// TIA Portal V19 export
FUNCTION "FC902_SafetyLogic" : Void   // FC902, F_LAD
{ S7_Optimized_Access := 'TRUE' }
// stored: AutoNumber false
BEGIN

REGION Network 1: Safety enabled to Robot Safemove
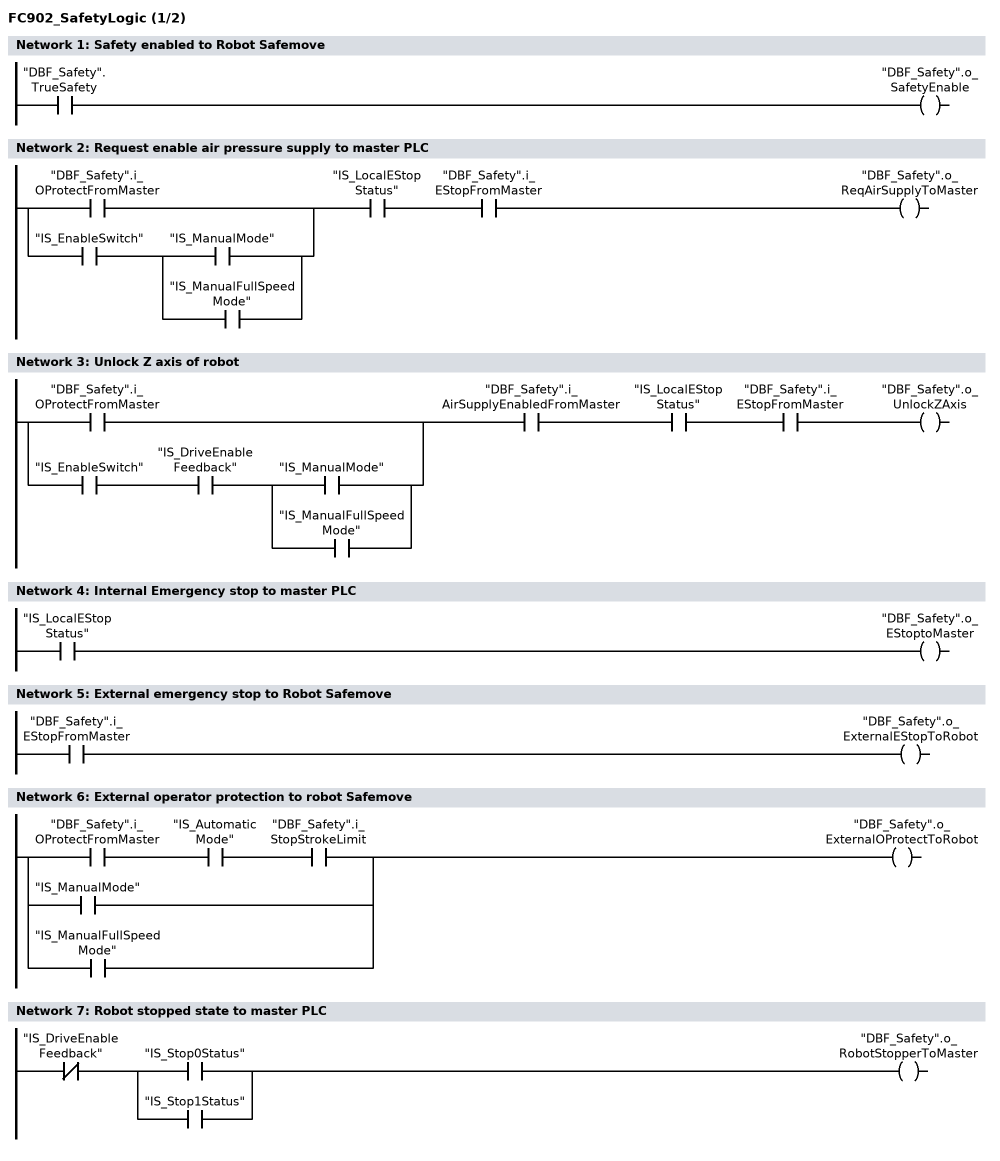
   RUNG wire#powerrail
      Contact( "DBF_Safety".TrueSafety )
      Coil( "DBF_Safety".o_SafetyEnable )
   END_RUNG
   // the same network as SCL:
   "DBF_Safety".o_SafetyEnable := "DBF_Safety".TrueSafety;
END_REGION

REGION Network 2: Request enable air pressure supply to master PLC
   RUNG wire#powerrail
      Contact( "DBF_Safety".i_OProtectFromMaster )
      wire#w1
      Contact( "IS_LocalEStopStatus" )
      Contact( "DBF_Safety".i_EStopFromMaster )
      Coil( "DBF_Safety".o_ReqAirSupplyToMaster )
   END_RUNG
   RUNG wire#powerrail
      Contact( "IS_EnableSwitch" )
      wire#w2
      Contact( "IS_ManualMode" )
   END_RUNG wire#w1
   RUNG wire#w2
      Contact( "IS_ManualFullSpeedMode" )
   END_RUNG wire#w1
   // the same network as SCL:
   "DBF_Safety".o_ReqAirSupplyToMaster := ("DBF_Safety".i_OProtectFromMaster OR ("IS_EnableSwitch" AND ("IS_ManualMode" OR "IS_ManualFullSpeedMode"))) AND "IS_LocalEStopStatus" AND "DBF_Safety".i_EStopFromMaster;
END_REGION

REGION Network 3: Unlock Z axis of robot
   RUNG wire#powerrail
      Contact( "DBF_Safety".i_OProtectFromMaster )
      wire#w1
      Contact( "DBF_Safety".i_AirSupplyEnabledFromMaster )
      Contact( "IS_LocalEStopStatus" )
      Contact( "DBF_Safety".i_EStopFromMaster )
      Coil( "DBF_Safety".o_UnlockZAxis )
   END_RUNG
   RUNG wire#powerrail
      Contact( "IS_EnableSwitch" )
      Contact( "IS_DriveEnableFeedback" )
      wire#w2
      Contact( "IS_ManualMode" )
   END_RUNG wire#w1
   RUNG wire#w2
      Contact( "IS_ManualFullSpeedMode" )
   END_RUNG wire#w1
   // the same network as SCL:
   "DBF_Safety".o_UnlockZAxis := ("DBF_Safety".i_OProtectFromMaster OR ("IS_EnableSwitch" AND "IS_DriveEnableFeedback" AND ("IS_ManualMode" OR "IS_ManualFullSpeedMode"))) AND "DBF_Safety".i_AirSupplyEnabledFromMaster AND "IS_LocalEStopStatus" AND "DBF_Safety".i_EStopFromMaster;
END_REGION

REGION Network 4: Internal Emergency stop to master PLC
   RUNG wire#powerrail
      Contact( "IS_LocalEStopStatus" )
      Coil( "DBF_Safety".o_EStoptoMaster )
   END_RUNG
   // the same network as SCL:
   "DBF_Safety".o_EStoptoMaster := "IS_LocalEStopStatus";
END_REGION

REGION Network 5: External emergency stop to Robot Safemove
   RUNG wire#powerrail
      Contact( "DBF_Safety".i_EStopFromMaster )
      Coil( "DBF_Safety".o_ExternalEStopToRobot )
   END_RUNG
   // the same network as SCL:
   "DBF_Safety".o_ExternalEStopToRobot := "DBF_Safety".i_EStopFromMaster;
END_REGION

REGION Network 6: External operator protection to robot Safemove
   RUNG wire#powerrail
      Contact( "DBF_Safety".i_OProtectFromMaster )
      Contact( "IS_AutomaticMode" )
      Contact( "DBF_Safety".i_StopStrokeLimit )
      wire#w1
      Coil( "DBF_Safety".o_ExternalOProtectToRobot )
   END_RUNG
   RUNG wire#powerrail
      Contact( "IS_ManualMode" )
   END_RUNG wire#w1
   RUNG wire#powerrail
      Contact( "IS_ManualFullSpeedMode" )
   END_RUNG wire#w1
   // the same network as SCL:
   "DBF_Safety".o_ExternalOProtectToRobot := ("DBF_Safety".i_OProtectFromMaster AND "IS_AutomaticMode" AND "DBF_Safety".i_StopStrokeLimit) OR "IS_ManualMode" OR "IS_ManualFullSpeedMode";
END_REGION

REGION Network 7: Robot stopped state to master PLC
   RUNG wire#powerrail
      I_Contact( "IS_DriveEnableFeedback" )
      wire#w1
      Contact( "IS_Stop0Status" )
      wire#w2
      Coil( "DBF_Safety".o_RobotStopperToMaster )
   END_RUNG
   RUNG wire#w1
      Contact( "IS_Stop1Status" )
   END_RUNG wire#w2
   // the same network as SCL:
   "DBF_Safety".o_RobotStopperToMaster := NOT "IS_DriveEnableFeedback" AND ("IS_Stop0Status" OR "IS_Stop1Status");
END_REGION

REGION Network 8: Power Off 24V Safety for FerRobotic
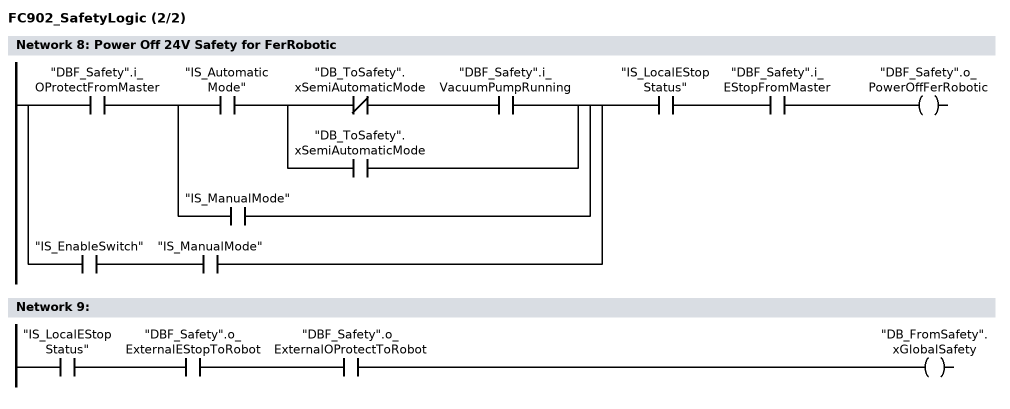
   RUNG wire#powerrail
      Contact( "DBF_Safety".i_OProtectFromMaster )
      wire#w1
      Contact( "IS_AutomaticMode" )
      wire#w2
      I_Contact( "DB_ToSafety".xSemiAutomaticMode )
      Contact( "DBF_Safety".i_VacuumPumpRunning )
      wire#w3
      Contact( "IS_LocalEStopStatus" )
      Contact( "DBF_Safety".i_EStopFromMaster )
      Coil( "DBF_Safety".o_PowerOffFerRobotic )
   END_RUNG
   RUNG wire#w2
      Contact( "DB_ToSafety".xSemiAutomaticMode )
   END_RUNG wire#w3
   RUNG wire#w1
      Contact( "IS_ManualMode" )
   END_RUNG wire#w3
   RUNG wire#powerrail
      Contact( "IS_EnableSwitch" )
      Contact( "IS_ManualMode" )
   END_RUNG wire#w3
   // the same network as SCL:
   "DBF_Safety".o_PowerOffFerRobotic := (("DBF_Safety".i_OProtectFromMaster AND (("IS_AutomaticMode" AND ((NOT "DB_ToSafety".xSemiAutomaticMode AND "DBF_Safety".i_VacuumPumpRunning) OR "DB_ToSafety".xSemiAutomaticMode)) OR "IS_ManualMode")) OR ("IS_EnableSwitch" AND "IS_ManualMode")) AND "IS_LocalEStopStatus" AND "DBF_Safety".i_EStopFromMaster;
END_REGION

REGION Network 9
   RUNG wire#powerrail
      Contact( "IS_LocalEStopStatus" )
      Contact( "DBF_Safety".o_ExternalEStopToRobot )
      Contact( "DBF_Safety".o_ExternalOProtectToRobot )
      Coil( "DB_FromSafety".xGlobalSafety )
   END_RUNG
   // the same network as SCL:
   "DB_FromSafety".xGlobalSafety := "IS_LocalEStopStatus" AND "DBF_Safety".o_ExternalEStopToRobot AND "DBF_Safety".o_ExternalOProtectToRobot;
END_REGION
END_FUNCTION
